// TIA Portal V20 export
// export: Created 2026-10-03T18:54:33.6329617Z, ExportSetting WithDefaults, DisplayName Totally Integrated Automation Portal, DisplayVersion V20 Update 4, DisplayName TIA Portal Openness, DisplayVersion V20 Update 4, DisplayName TIA Portal Version Control Interface, DisplayVersion V20 Update 4, DisplayName SINAMICS Startdrive Advanced, DisplayVersion V20 SP1 Update 1, DisplayName SINAMICS Startdrive G110M, G120, G120C, G120D, G120P, G115D, DisplayVersion V20 SP1 Update 1, DisplayName SINAMICS Startdrive G130, G150, S120, S150, SINAMICS MV, G220, S200, S210, DisplayVersion V20 SP1 Update 1, DisplayName STEP 7 Professional, DisplayVersion V20 Update 4, DisplayName STEP 7 Safety, DisplayVersion V20 Update 2, DisplayName WinCC Basic/Comfort/Advanced, DisplayVersion V20 Update 4, DisplayName WinCC Unified, DisplayVersion V20 Update 4
FUNCTION "SLC_COP_WORD" : Void   // FC1, SCL
TITLE = SLC COP (copy file) for B and N files
{ S7_Optimized_Access := 'TRUE' }
VERSION : 0.1
// Replaces COP #SrcFile:SrcElement #DstFile:DstElement Length for bit and integer files.
//  The converted data file DBs are numbered like the SLC files (N11 is DB11) and keep the SLC memory layout,
//  2 bytes per element, so the copy is a plain block copy between the two DBs.
// stored: AutoNumber true, IsIECCheckEnabled false, SetENOAutomatically false, UDAEnableTagReadback false
   VAR_INPUT
      SrcFile : DInt;   // Source data file number (11 for #N11:0)
      SrcElement : DInt;   // First source element (0 for #N11:0)
      DstFile : DInt;   // Destination data file number
      DstElement : DInt;   // First destination element
      Length : DInt;   // Number of elements to copy
   END_VAR
BEGIN
   // 16#84 is the DB memory area; each element is 2 bytes.
   POKE_BLK(area_src := 16#84, dbNumber_src := #SrcFile, byteOffset_src := #SrcElement * 2,
            area_dest := 16#84, dbNumber_dest := #DstFile, byteOffset_dest := #DstElement * 2,
            count := #Length * 2);
END_FUNCTION
